# EPICS SNL sequencer program: 2023/TestFunction/backup/epicsApp/liberaApp/src/StriplineHER.stt
program StriplineHER

%%#include <stdio.h>
%%#include <stdlib.h>
%%#include <assert.h>
%%#include <time.h>
%%#include <math.h>
%%#include <unistd.h>
%%#include "MT.h"

double X0, X1, Y, LM0, LM1, LM2,
/*--- HER (D8) ---*/
assign X0 to "TEST:X0";
assign X1 to "TEST:X1";
assign Y  to "TEST:Y";
assign LM1 to "TEST:LM0";
//assign LM2 to "TEST:LM1";
//assign LM3 to "TEST:LM2";

monitor X0;
monitor X1;
monitor LM0;
//monitor LM1;
//monitor LM2;

%{
  double x0;
  double x1;
  double y;
  double lm0;
  //double lm1;
  //double lm2;

  double Uniform(void)
  {
    return genrand_real3();
  }

  double rand_Lnormal(double mu, double sigma)
  {
    double y= mu + sigma*sqrt(-2.0*log(Uniform()))*sin(2.0*M_PI*Uniform());//gauss random number
    return y;
  }
}%

ss her_stripline {

  /*--- Initialization ---*/
  state init {
    when ()
    {
      pvGet(X0);
      pvGet(X1);
      //LM0 = Uniform();
      //LM1 = Uniform();
      //LM2 = Uniform();

      printf("StriplineHER initialization done.\n");

      %{
        init_genrand((unsigned)time(NULL));
      }%
    }
    state fit
  }

  /*--- Fit ---*/
  state fit {
    when ()
    {
      x0 = X0;
      x1 = X1;

      %{
	y = pow(X1 - 5.1/(4.*pow(M_PI,2.)) * pow(X0,2.) + 5./M_PI * X0 - 6., 2.) + 10 * (1. - 1./(8.*M_PI)) * cos(X0) + 10.
  + rand_Lnormal(0., 1.e-3);

      }%

      Y = y;
      pvPut(Y);

      LM0 = Uniform();
      pvPut(LM0);
      //pvPut(LM1);
      //pvPut(LM2);
      //pvPut(TH);

      %{
        usleep(0.1e+6);
      }%
    }
    state fit
  }
}
